TYPE E_Enum_2 :
(
	ZERO := 0,
	ONE := 1,
	TWO := 2,
	THREE := 3,
	THIRTEEN := 13,
	the_answer_to_life_the_universe_and_everything := 42
) INT;
END_TYPE

(* stored: Version 1.1.0.1, ProductVersion 3.1.4024.0
   DUT E_Enum_2: Id {5b2c3281-e8c6-4fff-add6-1b40d19b7459} *)
